// TIA Portal V16 export
// export: Created 2024-06-18T17:33:53.1762884Z, ExportSetting WithDefaults, DisplayName Totally Integrated Automation Portal, DisplayVersion V16, DisplayName TIA Portal Version Control Interface, DisplayVersion V16, DisplayName TIA Portal Openness, DisplayVersion V16, DisplayName STEP 7 Professional, DisplayVersion V16, DisplayName STEP 7 Safety, DisplayVersion V16, DisplayName WinCC Advanced, DisplayVersion V16
TYPE "Axis.RB_Memórias_Externas"
TITLE = Essa Memorias são escritas pelo software FORA do bloco do robô
// stored: IsFailsafeCompliant false
   STRUCT
      RB_Auxiliar_de_Programa : Array[1..32] of Bool;   // RB - Auxiliar de Programa 1 / Auxilia chamada de programa
      "RB_Aux_Aut.Trabalho" : Array[1..32] of Bool;   // Auxilia Autorização de Trabalho
      "RB_Aux_Aut.Intertravamento" : Array[1..32] of Bool;   // RB - Aux Liberação de Trabalho 1 / Auxilia Autorização de Intertravamento
      "RB_Aux_Rec.FimTrabalho" : Array[1..32] of Bool;   // RB - Aux Liberação de Trabalho 2 / Auxilia Reconhecimento Fim de Trabalho
   END_STRUCT;
END_TYPE
